{attribute 'qualified_only'}
{attribute 'strict'}
TYPE eErrorCodes : 
(
	AC_CONVEYOR_JAMMED := 16#101 , 
	AC_CONVEYOR_NOT_REACHED := 16#102,  
	AC_ET_USAGE_MEET := 16#201,
	AC_ET_SERIES_NG := 16#202
) UDINT;
END_TYPE
//  AC_CONVEYOR_JAMMED = '16#101'
//  AC_CONVEYOR_NOT_REACHED = '16#102'
//  AC_ET_USAGE_MEET = '16#201'
//  AC_ET_SERIES_NG = '16#202'

(* stored: Version 1.1.0.1, ProductVersion 3.1.4022.10
   EnumerationTextList eErrorCodes: Id {60e3e194-83de-45c5-919c-9caed3f38b0b} *)
